PROGRAM prgComEffIO
VAR
	fbCom		: FB_MqttCommunicator_V5;
END_VAR

fbCom(
	bConnect:= TRUE, 
	sUserName:= '795eb4ac-ab73-423a-978c-776b62a0fa2e', 
	sUserPassword:= 'f18add2b-7af7-4562-b9b6-6e5fd1b3afa3', 
	strAuthKey:= 'ENE87365342998', 
	eSavePositionCertificate:= eSavePositionOnPLC.ePostionC, 
	bConnected=> , 
	bError=> , 
	hrErrorCode=> , 
	eConnectionState=> , 
	eErrorMessage_Out=> );

END_PROGRAM

(* stored: Version 1.1.0.1, ProductVersion 3.1.4024.13
   POU prgComEffIO: Id {cbcd318b-bf51-484c-bcaa-d6efcdf43fe3}, SpecialFunc None *)
